Universal Robots PolyScope program: sequence.urp

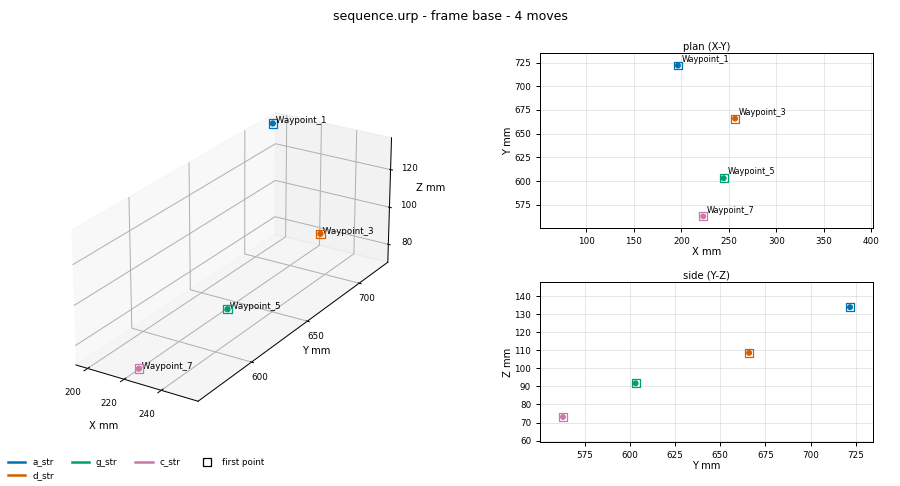
[picture p0: tool path of sequence.urp in frame base, 4 of 8 moves have a stored position in this frame; points joined in program order, loops and branches not executed]
Program sequence (installation=ext_control directory=/programs createdIn=5.17.3 lastSavedIn=5.17.3 robotSerialNumber=20245501435)
Calibrated DH parameters: a=[0.000154, -0.137004, -0.385524, -0.00002, 0.000092, 0]; d=[0.162441, 211.794786, -230.585024, 18.923638, 0.099786, 0.09951]; alpha=[1.569493, -0.001902, 0.003874, 1.570111, -1.570167, 0]; deltaTheta=[0, -1.242934, 1.056292, 0.186646, 0.000002, 0.000001]
InitVariablesNode
Robot Program (runOnlyOnce=false)
  Call a_str
  Call d_str
  Call g_str
  Call c_str
  Call g_str
  Call d_str
SubProgram -> a_str
SubProgram -> d_str
SubProgram -> g_str
SubProgram -> c_str
SubProgram a_str (keepSynchronizedWithDisk=false) programFile=/programs/a_str.urp
  MoveL speed 250 mm/s, acceleration 1200 mm/s^2 (useActiveTCP=true) feature=Base
    Waypoint Waypoint_1: TCP in base x=196.374 y=721.837 z=133.867 mm, rx=1.4747 ry=2.3846 rz=-1.033 rad; joints [-121.645, -30.465, 63.073, -81.878, -97.956, -145.045] deg; TCP offset x=28.21 y=-96.107 z=-99.69 mm, rx=0 ry=0 rz=0 rad
    Waypoint Waypoint_2 (Relative): relativeFromPosition TCP in base x=196.377 y=721.839 z=133.881 mm, rx=1.4747 ry=2.3846 rz=-1.033 rad; joints [-121.645, -30.466, 63.073, -81.877, -97.956, -145.045] deg; TCP in base x=519.54 y=370.1 z=282.791 mm, rx=-1.2592 ry=-2.2811 rz=1.5909 rad; joints [-159.63, -48.568, 76.17, -59.742, -121.226, -174.164] deg
SubProgram d_str (keepSynchronizedWithDisk=false) programFile=/programs/d_str.urp
  MoveL speed 250 mm/s, acceleration 1200 mm/s^2 (useActiveTCP=true) feature=Joint_6_name
    Waypoint Waypoint_3: TCP in base x=256.548 y=665.973 z=108.569 mm, rx=-1.5374 ry=-2.2292 rz=1.2496 rad; joints [-127.734, -31.287, 72.205, -80.819, -83.87, -151.225] deg; feature pose in base x=256.557 y=665.972 z=108.574 mm, rx=-1.5375 ry=-2.2292 rz=1.2495 rad
    Waypoint Waypoint_4 (Relative): relativeFromPosition TCP in base x=256.565 y=665.975 z=108.582 mm, rx=-1.5375 ry=-2.2292 rz=1.2495 rad; joints [-127.735, -31.288, 72.203, -80.818, -83.87, -151.225] deg; TCP in base x=308.201 y=212.166 z=168.469 mm, rx=1.5669 ry=2.3637 rz=-1.3134 rad; joints [-170.092, -63.301, 129.774, -117.857, -124.063, -180.489] deg; feature pose in base x=308.201 y=212.166 z=168.469 mm, rx=1.5669 ry=2.3637 rz=-1.3134 rad
SubProgram g_str (keepSynchronizedWithDisk=false) programFile=/programs/g_str.urp
  MoveL speed 250 mm/s, acceleration 1200 mm/s^2 (useActiveTCP=true) feature=Base
    Waypoint Waypoint_5: TCP in base x=244.537 y=603.172 z=91.747 mm, rx=-1.7467 ry=-2.0948 rz=0.8077 rad; joints [-130.747, -35.867, 89.817, -110.043, -73.974, -145.761] deg
    Waypoint Waypoint_6 (Relative): relativeFromPosition TCP in base x=244.521 y=603.182 z=91.749 mm, rx=-1.7467 ry=-2.0948 rz=0.8077 rad; joints [-130.745, -35.867, 89.817, -110.044, -73.975, -145.76] deg; TCP in base x=300.327 y=207.838 z=8.82 mm, rx=-1.2367 ry=-1.7305 rz=1.136 rad; joints [-170.03, -34.371, 126.934, -113.556, -94.765, -185.278] deg
SubProgram c_str (keepSynchronizedWithDisk=false) programFile=/programs/c_str.urp
  MoveL speed 250 mm/s, acceleration 1200 mm/s^2 (useActiveTCP=true) feature=Base
    Waypoint Waypoint_7: TCP in base x=222.973 y=562.956 z=73.09 mm, rx=-1.7404 ry=-1.5254 rz=0.3572 rad; joints [-130.567, -31.955, 101.515, -146.824, -42.301, -128.37] deg
    Waypoint Waypoint_8 (Relative): relativeFromPosition TCP in base x=225.604 y=562.943 z=77.706 mm, rx=-1.7406 ry=-1.5243 rz=0.3485 rad; joints [-130.763, -32.421, 101.483, -146.672, -42.264, -128.37] deg; TCP in base x=108.241 y=170.343 z=-59.719 mm, rx=-1.3852 ry=-1.4777 rz=0.7367 rad; joints [-170.461, -4.85, 143.353, -161.62, -71.094, -186.243] deg
